# EPICS autosave request: PIpiezo/E725_settings.req
$(P)$(Q):WFSETUP:WR
$(P)$(Q):WFSTART:WR
$(P)$(Q):WFSTOP:WR
